TYPE csp_case_feed_kinematic_status_enum :
(
	CSP_CASE_FEED_KINEMATIC_STATUS_NOT_INITIALIZED 							:= 0,
	CSP_CASE_FEED_KINEMATIC_STATUS_DISABLED 								:= 10,
	CSP_CASE_FEED_KINEMATIC_STATUS_ENABLE_REQUEST 							:= 20,
	CSP_CASE_FEED_KINEMATIC_STATUS_ENABLING 								:= 30,
	CSP_CASE_FEED_KINEMATIC_STATUS_ENABLED 									:= 40,
	CSP_CASE_FEED_KINEMATIC_STATUS_CHANGE_OVER_MODE                         := 50,
    CSP_CASE_FEED_KINEMATIC_STATUS_CHANGE_OVER_MODE_DONE                    := 60,   	
	CSP_CASE_FEED_KINEMATIC_STATUS_KIN_CONFIG								:= 100,
	CSP_CASE_FEED_KINEMATIC_STATUS_JOG_ACS1									:= 101,
	CSP_CASE_FEED_KINEMATIC_STATUS_JOG_ACS2									:= 102,
	CSP_CASE_FEED_KINEMATIC_STATUS_JOG_ACS3									:= 103,
	CSP_CASE_FEED_KINEMATIC_STATUS_JOG_MCS1									:= 105,
	CSP_CASE_FEED_KINEMATIC_STATUS_JOG_MCS2									:= 106,
	CSP_CASE_FEED_KINEMATIC_STATUS_JOG_MCS3									:= 107,
	CSP_CASE_FEED_KINEMATIC_STATUS_MOVE_ACS1								:= 111,
	CSP_CASE_FEED_KINEMATIC_STATUS_MOVE_ACS2								:= 112,
	CSP_CASE_FEED_KINEMATIC_STATUS_MOVE_ACS3								:= 113,
	CSP_CASE_FEED_KINEMATIC_STATUS_MOVE_MCS1								:= 115,
	CSP_CASE_FEED_KINEMATIC_STATUS_MOVE_MCS2								:= 116,
	CSP_CASE_FEED_KINEMATIC_STATUS_MOVE_MCS3								:= 117,
	CSP_CASE_FEED_KINEMATIC_STATUS_STOP_ACS1								:= 121,
	CSP_CASE_FEED_KINEMATIC_STATUS_STOP_ACS2								:= 122,
	CSP_CASE_FEED_KINEMATIC_STATUS_STOP_ACS3								:= 123,
	CSP_CASE_FEED_KINEMATIC_STATUS_STOP_MCS1								:= 125,
	CSP_CASE_FEED_KINEMATIC_STATUS_STOP_MCS2								:= 126,
	CSP_CASE_FEED_KINEMATIC_STATUS_STOP_MCS3								:= 127,		
	CSP_CASE_FEED_KINEMATIC_STATUS_PHASE_REQUEST							:= 150,
	CSP_CASE_FEED_KINEMATIC_STATUS_PHASING									:= 160,
	CSP_CASE_FEED_KINEMATIC_STATUS_PHASED									:= 170,
	CSP_CASE_FEED_KINEMATIC_STATUS_READY_TO_ENGAGE							:= 180,
	CSP_CASE_FEED_KINEMATIC_STATUS_CAM_ENGAGED_REQ							:= 200,	
	CSP_CASE_FEED_KINEMATIC_STATUS_CAM_ENGAGED								:= 210,
	CSP_CASE_FEED_KINEMATIC_STATUS_STOP_REQUEST 							:= 500,
	CSP_CASE_FEED_KINEMATIC_STATUS_DISABLE_REQUEST 							:= 510,
	CSP_CASE_FEED_KINEMATIC_STATUS_DISABLING_KINEMATIC						:= 511,
	CSP_CASE_FEED_KINEMATIC_STATUS_DISABLING_AXIS							:= 512,
	CSP_CASE_FEED_KINEMATIC_STATUS_DISABLING 								:= 520		
) := CSP_CASE_FEED_KINEMATIC_STATUS_NOT_INITIALIZED;
END_TYPE

(* stored: Version 1.1.0.1, ProductVersion 3.1.4022.12
   DUT csp_case_feed_kinematic_status_enum: Id {d11c499c-6ef2-4717-a9af-e1bd75a756b3} *)
